PROGRAM MAIN
VAR
END_VAR

END_PROGRAM

(* stored: Version 1.1.0.1
   POU MAIN: Id {8b4d3fc1-5859-418d-99c5-adaab40edce7} *)
